FUNCTION TryConvert_REAL_TO_REAL : BOOL
VAR_INPUT
	in : REAL;
	out : REFERENCE TO REAL;
END_VAR

out := in;
TryConvert_REAL_TO_REAL := TRUE;

END_FUNCTION

(* stored: Version 1.1.0.1, ProductVersion 3.1.4024.12
   POU TryConvert_REAL_TO_REAL: Id {e9f57f16-740c-444f-bd51-74bee7080bdc}, SpecialFunc None *)
